FUNCTION_BLOCK Section0
  (* Standard: 61499-2 *)
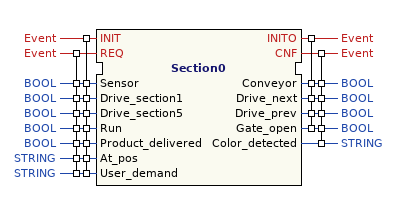
  EVENT_INPUT
    INIT WITH Sensor, Drive_section1, Drive_section5, Run, Product_delivered, At_pos, User_demand;
    REQ WITH Sensor, Drive_section1, Drive_section5, Run, Product_delivered, At_pos, User_demand;
  END_EVENT
  EVENT_OUTPUT
    INITO WITH Conveyor, Drive_next, Drive_prev, Gate_open;
    CNF WITH Conveyor, Drive_next, Drive_prev, Gate_open, Color_detected;
  END_EVENT
  VAR_INPUT
    Sensor : BOOL;
    Drive_section1 : BOOL;
    Drive_section5 : BOOL;
    Run : BOOL;
    Product_delivered : BOOL;
    At_pos : STRING;
    User_demand : STRING;
  END_VAR
  VAR_OUTPUT
    Conveyor : BOOL;
    Drive_next : BOOL;
    Drive_prev : BOOL;
    Gate_open : BOOL;
    Color_detected : STRING;
  END_VAR
  FBS
    FB1 : DisableConveyor;
    FB3 : ;
    FB5 : E_R_TRIG;
    FB4 : ;
    FB6 : E_MERGE;
    FB7 : E_MERGE;
    FB8 : ;
    FB9 : E_MERGE;
    FB2 : Section0Ctrl;
  END_FBS
  EVENT_CONNECTIONS
    INIT TO FB2.INIT;
    REQ TO FB6.EI1;
    FB2.CNF TO FB1.REQ;
    FB2.INITO TO FB1.INIT;
    REQ TO FB1.REQ;
    INIT TO FB3.null;
    FB2.CNF TO FB5.EI;
    FB5.EO TO FB3.null;
    FB3.null TO FB3.null;
    FB3.null TO FB4.null;
    FB4.null TO FB6.EI2;
    FB6.EO TO FB9.EI2;
    FB1.CNF TO FB7.EI1;
    FB3.null TO FB7.EI2;
    FB7.EO TO CNF;
    REQ TO FB4.null;
    REQ TO FB8.null;
    FB9.EO TO FB2.REQ;
    FB8.null TO FB9.EI1;
  END_CONNECTIONS
  DATA_CONNECTIONS
    Run TO FB1.QI;
    Sensor TO FB2.Sensor;
    Drive_section5 TO FB2.Drive_section5;
    Product_delivered TO FB2.Product_delivered;
    FB2.Conveyor TO FB1.ConvIn;
    FB2.Drive_next TO Drive_next;
    FB2.Drive_prev TO Drive_prev;
    FB2.Gate_open TO Gate_open;
    FB1.ConvOut TO Conveyor;
    Drive_section1 TO FB2.Drive_section1;
    FB2.Check_color TO FB5.QI;
    User_demand TO FB4.null;
    FB3.null TO FB4.null;
    FB4.null TO FB2.Valid_product;
    FB3.null TO Color_detected;
    At_pos TO FB8.null;
    FB8.null TO FB2.Robotino_docked;
  END_CONNECTIONS
END_FUNCTION_BLOCK
